// TIA Portal V20 export
// export: Created 2026-04-28T10:17:59.1070244Z, ExportSetting WithDefaults, DisplayName Totally Integrated Automation Portal, DisplayVersion V20, DisplayName TIA Portal Openness, DisplayVersion V20, DisplayName TIA Portal Version Control Interface, DisplayVersion V20, DisplayName SINAMICS Startdrive Advanced, DisplayVersion V20, DisplayName SINAMICS Startdrive G130, G150, S120, S150, SINAMICS MV, G220, S200, S210, DisplayVersion V20, DisplayName SINAMICS Startdrive G110M, G120, G120C, G120D, G120P, G115D, DisplayVersion V20, DisplayName STEP 7 Professional, DisplayVersion V20, DisplayName STEP 7 Safety, DisplayVersion V20, DisplayName WinCC Basic/Comfort/Advanced, DisplayVersion V20, DisplayName WinCC Unified, DisplayVersion V20
TYPE "Daten_SPT_40"
// stored: IsFailsafeCompliant false
   STRUCT
      xFlyFire : Bool := false;   // Selection Flying Fire
      xBarrelxx : Bool := false;   // Selection Barrel
      xReturn : Bool := false;   // Selection return
      xPrede : Bool := false;   // Selection Dust conveying fan
      xPredeIst : Bool := false;   // Selection Dust conveying fan Actual Value
      xPredeSoll : Bool := false;   // Selection Dust conveying fan Set value
      RangePrede : DInt := 0;   // Range Dust conveying fan
      txt_rPrede : DInt := 0;   // Set value Dust conveying fan
      iTakt_Prede : DInt := 0;   // Interval for recording the measured values
      iAnzWerte_Prede : DInt := 0;   // Number of measured values
      xDiDuFiBa : Bool := false;   // Selection Differential pressure filter dust return
      txt_rDiDuFiBa : DInt := 0;   // Alarm Value Differential pressure filter dust return
      txt_max_rDiDuFiBa : DInt := 0;   // Input Value Limit Differential pressure filter dust return
      RangeDiDuFiBa : DInt := 0;   // Range Differential pressure filter dust return
      iTakt_DiDuFiBa : DInt := 0;   // Interval for recording the measured values
      iAnzWerte_DiDuFiBa : DInt := 0;   // Number of measured values
      xCyclone : Bool := false;   // Selection Cyclone
      txt_rCyclone : DInt := 0;   // Selection Cyclone 1 or 2
      xRet_Bin : Bool := false;   // Selection Return/Bin
      txt_rReturn : DInt := 0;   // Return or Bin
      xKnVa40 : Bool := false;   // Knocker valves cyclone
      t_iKnValve_1 : Time := T#0MS;   // Knock Valve on, Cyklon
      t_iKnBreake_1 : Time := T#0MS;   // Knock Valve Breake, Cyklon
      xRotaryFeeder : Bool := false;   // Selection Rotary Feeder
      xFlRaAirPrede : Bool := false;   // Selection Volume flow dust return
      RangeFlRaAirPrede : DInt := 0;   // Range Volume flow dust return
      xTempPrede : Bool := false;   // Selection Feed temperature dust return
      RangeTempPrede : DInt := 0;   // Range Feed temperature dust return
      iTakt_FlRaAirPrede : DInt := 0;   // Interval for recording the measured values
      iAnzWerte_FlRaAirPrede : DInt := 0;   // Number of measured values
      iTakt_TempPrede : DInt := 0;   // Interval for recording the measured values
      iAnzWerte_TempPrede : DInt := 0;   // Number of measured values
      xVibLimitSw_40 : Bool := 0;   // Dust container fill level
      xPrede_Man : Bool := false;   // Selection Dust conveyor fan manual
      xprede_ohneweiche : Bool := false;   // Switch with /without
      xOptKnVa : Bool := false;   // Knocker valves automatically
      xCyFillingMax_Option : Bool;   // Selection Cyclone Container Fill Level Max. 0=without, 1=with
      xFlRaCy_Option : Bool;   // Selection Cyclone flow monitoring dust return 0=without, 1=with
      RangeFlRaCy : DInt;   // Range Cyclone flow monitoring dust return
      iTakt_FlRaCy : DInt;   // Interval for recording the measured values
      iAnzWerte_FlRaCy : DInt;   // Number of measured values
      txt_rFlRaCy : DInt;   // Max. Value Cyclone flow monitoring dust return
   END_STRUCT;
END_TYPE
